TYPE ST_RecipeTypeMachine :
STRUCT
	// Test Line High Level Structure
	nIdx	: UINT;
	bEnable	: BOOL;
	nActiveStationCount	: UINT;
END_STRUCT
END_TYPE

(* stored: Version 1.1.0.1
   DUT ST_RecipeTypeMachine: Id {785538c5-51ee-0afe-2459-d6a2533faecf} *)
